FUNCTION_BLOCK FB_HomingTimer
VAR_OUTPUT
	Done : BOOL;
END_VAR
VAR
	i			: LINT := 0;
	LoopCount	: LINT;
END_VAR


Done := False;

i := i + 1;

IF i >= LoopCount THEN
	Done := TRUE;
END_IF

METHOD FB_init : BOOL
VAR_INPUT
	bInitRetains : BOOL; // if TRUE, the retain variables are initialized (warm start / cold start)
	bInCopyCode : BOOL;  // if TRUE, the instance afterwards gets moved into the copy code (online change)
	
	LoopsToRun	: LINT;
END_VAR

THIS^.i := 0;
THIS^.LoopCount := LoopsToRun;
END_METHOD

END_FUNCTION_BLOCK

(* stored: Version 1.1.0.1, ProductVersion 3.1.4022.17
   POU FB_HomingTimer: Id {6daf19c6-1dde-4928-a084-d0c6759bf0ba}, SpecialFunc None
   Method FB_init: Id {e2775d28-756d-4453-b544-630b65051fee} *)
